{attribute 'qualified_only'}
{attribute 'strict'}
TYPE E_IO2_Type :
(
	BLOCKED	:= 0,
	NO := 1,
	NC := 2
);
END_TYPE

(* stored: Version 1.1.0.1
   DUT E_IO2_Type: Id {e68513ab-47e5-48b0-bfcf-e15080969b49} *)
